FUNCTION_BLOCK FB_MagnetPermIntlk
VAR_INPUT
	SystemPermIntlkOK				: BOOL;
END_VAR
VAR_OUTPUT
	bMagnetCmdOn						: BOOL;
END_VAR
VAR
	MagnetPermIntlkOK				: BOOL;
	nForCounterDiverting		: UDINT;
	ftPermIntlk					: Tc2_Standard.F_TRIG;
END_VAR

//Command Diverting to Magnet for any designated mover
FOR nForCounterDiverting := GC.nNumMinMovers TO GVL_General.nNumMovers DO

	MagnetPermIntlkOK	:= SystemPermIntlkOK AND
		fbPlanarXtsMover[nForCounterDiverting].P_MoverStatus.CommandedToDivert AND
		(TrackSectors[nForCounterDiverting].SingularSectorStatus[GC.SHORTCUT_MAIN_SECTOR_IPART].MoverCountOnSector <
			GVL_General.stSwitchConfig.SwitchModeInternal.MaxAllowedCountOnShortcut);
			
	IF MagnetPermIntlkOK AND_THEN 
		GVL_Mc3.TrackSectors[nForCounterDiverting].SingularSectorStatus[GC.MAG_ON_SECTOR_OPART].MoverIsOnSector THEN
		bMagnetCmdOn := TRUE;
//		EXIT;
	ELSIF ftPermIntlk.Q OR GVL_Mc3.TrackSectors[nForCounterDiverting].SingularSectorStatus[GC.MAG_ON_SECTOR_OPART].MoverExitedSector.Q THEN
		fbPlanarXtsMover[nForCounterDiverting].P_CmdDivert 	:= FALSE;
		fbPlanarXtsMover[nForCounterDiverting].P_MoverStatus.IntervalMarked	:= FALSE;
		bMagnetCmdOn := FALSE;
	END_IF
	
//	IF TrackSectors[nForCounterDiverting].SingularSectorStatus[GC.SHORTCUT_DIVERT_SECTOR_IPART].MoverExitedSector.Q THEN
//			fbPlanarXtsMover[nForCounterDiverting].P_MoverStatus.IntervalMarked		:= FALSE;
//	END_IF

END_FOR

ftPermIntlk(CLK := MagnetPermIntlkOK);

PROPERTY P_OK : REFERENCE TO BOOL
GET
P_OK REF= MagnetPermIntlkOK;
END_GET
END_PROPERTY

END_FUNCTION_BLOCK

(* stored: Version 1.1.0.1
   POU FB_MagnetPermIntlk: Id {962a6221-0f3e-03bc-045d-7d19eb7395ad}, SpecialFunc None
   Property P_OK: Id {fc7fc1bf-2e5f-0caa-35f3-e55afb89eca7}
   Get Get: Id {0e6c77fc-4f91-0be7-2897-0cbafedb3e53} *)
